// TIA Portal project "ModbusTCP_S7-1500" (V18)
// Test del protocolo Modbus TCP usando MB_Server y QModMaster

(* hardware
DEVICE "S7-1500/ET200MP station_1"  S7-1500 station
   slot 0: "Rail_0"  Rack  6ES7 590-1***0-0AA0
   slot 1: "PLC_1"  CPU 1511-1 PN  6ES7 511-1AL03-0AB0  V3.0
      slot 3: "CPU display_1"  6ES7591-1AA00-0AA0
      slot 32768: "PROFINET interface_1"  X1
         slot 32769: "Port_1"  X1 P1
         slot 32770: "Port_2"  X1 P2
      slot 34817: "Virtual CP interface port_1"  Virtual CP interface port  Virtual CP interface port
*)

// ===== PLC "PLC_1"  CPU 1511-1 PN =====

VAR_GLOBAL   // PLC tag table "Default tag table"
   "start" AT %I0.0 : Bool;
   "stop" AT %I0.1 : Bool;
   "motor" AT %Q0.0 : Bool;
   "System_Byte" AT %MB1 : Byte;
   "FirstScan" AT %M1.0 : Bool;
   "DiagStatusUpdate" AT %M1.1 : Bool;
   "AlwaysTRUE" AT %M1.2 : Bool;
   "AlwaysFALSE" AT %M1.3 : Bool;
   "System_Byte(1)" AT %MB1 : Byte;
   "Clock_Byte" AT %MB0 : Byte;
   "Clock_10Hz" AT %M0.0 : Bool;
   "Clock_5Hz" AT %M0.1 : Bool;
   "Clock_2.5Hz" AT %M0.2 : Bool;
   "Clock_2Hz" AT %M0.3 : Bool;
   "Clock_1.25Hz" AT %M0.4 : Bool;
   "Clock_1Hz" AT %M0.5 : Bool;
   "Clock_0.625Hz" AT %M0.6 : Bool;
   "Clock_0.5Hz" AT %M0.7 : Bool;
   "Alarma_1" AT %M100.0 : Bool;
   "Tag_1" AT %MW28 : Word;
   "Tag_2" AT %MW30 : Word;
   "Tag_3" AT %MW38 : Word;
   "Tag_4" AT %MW48 : Word;
   "Tag_5" AT %MW50 : Word;
   "Tag_6" AT %MW86 : Word;
   "Tag_7" AT %MW88 : Word;
   "Tag_8" AT %MW90 : Word;
END_VAR

DATA_BLOCK "Modbus_Data"   // DB1
{ S7_Optimized_Access := 'FALSE' }
VERSION : 0.1
   VAR
      Data_Array : Array[0..119] of UInt;
   END_VAR
BEGIN
   // Data_Array[52] : ALARMA W52: 0: Emergencia, 1: Térmico motor, 2: Falta fase
   // Data_Array[53] : ALARMA W53
   // Data_Array[54] : ALARMA W54
   // Data_Array[55] : ALARMA W55
END_DATA_BLOCK

DATA_BLOCK "Modbus_Config"   // DB2
{ S7_Optimized_Access := 'TRUE' }
VERSION : 0.1
   VAR
      Config : TCON_IP_v4;
   END_VAR
BEGIN
   Config.InterfaceId := 64;
   Config.ID := 16#1;
   Config.ConnectionType := 16#0B;
   Config.LocalPort := 502;
END_DATA_BLOCK

DATA_BLOCK "SCADA_Comm"   // DB4
{ S7_Optimized_Access := 'FALSE' }
VERSION : 0.1
   VAR
      cmd_Start : Bool;
      cmd_Stop : Bool;
      sts_Motor : Bool;
   END_VAR
BEGIN
END_DATA_BLOCK

DATA_BLOCK "FB_Alarmas1_DB"   // DB5
{ S7_Optimized_Access := 'TRUE' }
VERSION : 0.1
// stored: InstanceOfName FB_Alarmas
"FB_Alarmas"
BEGIN
END_DATA_BLOCK

DATA_BLOCK "FB_Alarmas2_DB"   // DB6
{ S7_Optimized_Access := 'TRUE' }
VERSION : 0.1
// stored: InstanceOfName FB_Alarmas
"FB_Alarmas"
BEGIN
END_DATA_BLOCK

DATA_BLOCK "FB_Sim_Produccion_DB"   // DB7
{ S7_Optimized_Access := 'TRUE' }
VERSION : 0.1
// stored: InstanceOfName FB_Sim_Produccion
"FB_Sim_Produccion"
BEGIN
END_DATA_BLOCK

DATA_BLOCK "FB_SIM_Produccion_V2_DB"   // DB8
{ S7_Optimized_Access := 'TRUE' }
VERSION : 0.1
// stored: InstanceOfName FB_SIM_Produccion_V2
"FB_SIM_Produccion_V2"
BEGIN
END_DATA_BLOCK

FUNCTION_BLOCK "FB_Alarmas"   // FB1, SCL
{ S7_Optimized_Access := 'TRUE' }
VERSION : 0.1
   VAR_INPUT
      i_Bit_0 : Bool;
      i_Bit_1 : Bool;
      i_Bit_2 : Bool;
      i_Bit_3 : Bool;
      i_Bit_4 : Bool;
      i_Bit_5 : Bool;
      i_Bit_6 : Bool;
      i_Bit_7 : Bool;
      i_Bit_8 : Bool;
      i_Bit_9 : Bool;
      i_Bit_10 : Bool;
      i_Bit_11 : Bool;
      i_Bit_12 : Bool;
      i_Bit_13 : Bool;
      i_Bit_14 : Bool;
      i_Bit_15 : Bool;
      i_Reset : Bool;   // Entrada del botón de reset
   END_VAR
   VAR_OUTPUT
      o_Bit_0 : Bool;
      o_Bit_1 : Bool;
      o_Bit_2 : Bool;
      o_Bit_3 : Bool;
      o_Bit_4 : Bool;
      o_Bit_5 : Bool;
      o_Bit_6 : Bool;
      o_Bit_7 : Bool;
      o_Bit_8 : Bool;
      o_Bit_9 : Bool;
      o_Bit_10 : Bool;
      o_Bit_11 : Bool;
      o_Bit_12 : Bool;
      o_Bit_13 : Bool;
      o_Bit_14 : Bool;
      o_Bit_15 : Bool;
      enAlarma : Bool;
   END_VAR
BEGIN
   // 1. Construcción de la palabra de alarmas actual
   // 3. Gestión de la salida
   // Si doy reset, la palabra de salida se pone a cero, sino refleja los bits de entrada.
   IF #i_Reset THEN
       // 1. Construcción de la palabra de alarmas actual
       #o_Bit_0 := 0;
       #o_Bit_1 := 0;
       #o_Bit_2 := 0;
       #o_Bit_3 := 0;
       #o_Bit_4 := 0;
       #o_Bit_5 := 0;
       #o_Bit_6 := 0;
       #o_Bit_7 := 0;
       #o_Bit_8 := 0;
       #o_Bit_9 := 0;
       #o_Bit_10 := 0;
       #o_Bit_11 := 0;
       #o_Bit_12 := 0;
       #o_Bit_13 := 0;
       #o_Bit_14 := 0;
       #o_Bit_15 := 0;
   ELSE
       // 1. Construcción de la palabra de alarmas actual
       #o_Bit_0 := #i_Bit_0;
       #o_Bit_1 := #i_Bit_1;
       #o_Bit_2 := #i_Bit_2;
       #o_Bit_3 := #i_Bit_3;
       #o_Bit_4 := #i_Bit_4;
       #o_Bit_5 := #i_Bit_5;
       #o_Bit_6 := #i_Bit_6;
       #o_Bit_7 := #i_Bit_7;
       #o_Bit_8 := #i_Bit_8;
       #o_Bit_9 := #i_Bit_9;
       #o_Bit_10 := #i_Bit_10;
       #o_Bit_11 := #i_Bit_11;
       #o_Bit_12 := #i_Bit_12;
       #o_Bit_13 := #i_Bit_13;
       #o_Bit_14 := #i_Bit_14;
       #o_Bit_15 := #i_Bit_15;
   END_IF;

   // Esto sigue siendo un poco largo pero es más limpio que un IF
   #enAlarma := #o_Bit_0 OR #o_Bit_1 OR #o_Bit_2 OR #o_Bit_3 OR
   #o_Bit_4 OR #o_Bit_5 OR #o_Bit_6 OR #o_Bit_7 OR
   #o_Bit_8 OR #o_Bit_9 OR #o_Bit_10 OR #o_Bit_11 OR
   #o_Bit_12 OR #o_Bit_13 OR #o_Bit_14 OR #o_Bit_15;

   // -------------------------------------------------------------
END_FUNCTION_BLOCK

FUNCTION_BLOCK "FB_Sim_Produccion"   // FB2, SCL
{ S7_Optimized_Access := 'TRUE' }
VERSION : 0.1
   VAR_INPUT
      IntervaloS : Time :=  T#1M;   // Intervalo de muestreo >> Escribe aquí T#1M o T#15M
   END_VAR
   VAR
      tCiclo : TON_TIME;   // Timer interno
      Seed : UDInt := 123456;   // Semilla aleatoria inicial
      Golpes : Int := 0;   // Estas variables son ESTÁTICAS: Se guardan solas en el DB de Instancia
   END_VAR
   VAR_TEMP
      valInt : Int;
   END_VAR
BEGIN
   // ============================================================
   // FB_Sim_Produccion — Versión Function Block (FB)
   // Simulación de datos de producción para SCADA Node3
   // ============================================================

   // 1. Temporizador cíclico
   #tCiclo(IN := NOT #tCiclo.Q, PT := #IntervaloS);

   // Lógica ejecutada en cada pulso del timer
   IF #tCiclo.Q THEN

       // --- SIMULACIÓN ALEATORIA ---

       // W14: TEMP_SP_SUP (180-220)
       #Seed := #Seed * 1664525 + 1013904223;
       #valInt := 180 + UDINT_TO_INT(#Seed MOD 41);
       "Tag_1" := #valInt;

       // W15: TEMP_SP_INF (160-200)
       #Seed := #Seed * 1664525 + 1013904223;
       #valInt := 160 + UDINT_TO_INT(#Seed MOD 41);
       "Tag_2" := #valInt;

       // W19: CONSUMO kW (10-25)
       #Seed := #Seed * 1664525 + 1013904223;
       #valInt := 10 + UDINT_TO_INT(#Seed MOD 16);
       "Tag_3" := #valInt;

       // W24: TEMP REAL SUP
       #Seed := #Seed * 1664525 + 1013904223;
       #valInt := 200 + UDINT_TO_INT(#Seed MOD 11) - 5;
       "Tag_4" := #valInt;

       // W25: TEMP REAL INF
       #Seed := #Seed * 1664525 + 1013904223;
       #valInt := 180 + UDINT_TO_INT(#Seed MOD 11) - 5;
       "Tag_5" := #valInt;

       // W43: ESTADO (0=Stop, 1=Run, 2=Alarma)
       #Seed := #Seed * 1664525 + 1013904223;
       #valInt := UDINT_TO_INT(#Seed MOD 3);
       "Tag_6" := #valInt;

       // W44: TIEMPO CICLO (8-12s)
       #Seed := #Seed * 1664525 + 1013904223;
       #valInt := 8 + UDINT_TO_INT(#Seed MOD 5);
       "Tag_7" := #valInt;

       // W45: CONTADOR GOLPES (Sumamos 5-20)
       #Seed := #Seed * 1664525 + 1013904223;
       #Golpes := #Golpes + 5 + UDINT_TO_INT(#Seed MOD 16);
       "Tag_8" := #Golpes;

   END_IF;
END_FUNCTION_BLOCK

FUNCTION_BLOCK "FB_SIM_Produccion_V2"   // FB3, SCL
{ S7_Optimized_Access := 'TRUE' }
VERSION : 0.1
   VAR_INPUT
      Enable : Bool := TRUE;
      IntervaloS : Time := T#1M;   // El contador suma cada este tiempo
   END_VAR
   VAR_OUTPUT
      outSPSup : Int;   // Conectar a W14 (%MW28)
      outSPInf : Int;   // Conectar a W15 (%MW30)
      outConsumo : Int;   // Conectar a W19 (%MW38)
      outTempSup : Int;   // Conectar a W24 (%MW48)
      outTempInf : Int;   // Conectar a W25 (%MW50)
      outCiclo : Int;   // Conectar a W44 (%MW88)
      outGolpes : Int;   // Conectar a W45 (%MW90)
   END_VAR
   VAR
      tCiclo : TON_TIME;   // Timer interno
      Seed : UDInt := 54321;   // Semilla aleatoria
      GolpesAcum : Int;   // Memoria interna de producción
      CicloUltimo : Int := 10;   // Valor inicial para que no empiece en 0
      PrimerScan : Bool := TRUE;
   END_VAR
   VAR_TEMP
      valInt : Int;
   END_VAR
BEGIN
   // ============================================================
   // FB_Sim_Produccion_V3 — Versión con Salidas Parametrizables
   // ============================================================
   (*
   Pin de Salida   Registro    Modbus PLC (Sugerido)  Descripción
   #outSPSup       W14 %MW28   SetPoint               Temp Superior
   outSPInf        W15 %MW30   SetPoint               Temp Inferior
   outConsumo      W19 %MW38   Consumo (kW)
   outTempSup      W24 %MW48   Temp Real Superior
   outTempInf      W25 %MW50   Temp Real Inferior
   outCiclo        W44 %MW88   Tiempo de Ciclo
   outGolpes       W45 %MW90   Contador de Producción
   *)

   // ============================================================
   // FB_Sim_Produccion_V7 — Versión Permanente (Salidas fijas)
   // ============================================================
   // 1. Temporizador
   #tCiclo(IN := #Enable AND NOT #tCiclo.Q,
           PT := #IntervaloS);

   IF NOT #Enable THEN
       RETURN;
   END_IF;

   // 2. CÁLCULO DE VALORES DINÁMICOS (Cada scan)
   #Seed := #Seed * 1664525 + 1013904223;

   #outSPSup := 200 + UDINT_TO_INT(#Seed MOD 3) - 1;
   #outSPInf := 180 + UDINT_TO_INT((#Seed / 10) MOD 3) - 1;
   #outTempSup := 198 + UDINT_TO_INT((#Seed / 100) MOD 5);
   #outTempInf := 178 + UDINT_TO_INT((#Seed / 1000) MOD 5);
   #outConsumo := 20 + UDINT_TO_INT((#Seed / 50) MOD 2);

   // 3. LÓGICA DE INCREMENTO (Solo cuando el timer da el pulso)
   IF #tCiclo.Q OR #PrimerScan THEN
       #GolpesAcum := #GolpesAcum + 1;
       #CicloUltimo := 8 + UDINT_TO_INT(#Seed MOD 5);
       #PrimerScan := FALSE;
   END_IF;

   // 4. ASIGNACIÓN PERMANENTE (Fuera del IF para que nunca sea cero)
   #outGolpes := #GolpesAcum;
   #outCiclo := #CicloUltimo;
END_FUNCTION_BLOCK

ORGANIZATION_BLOCK "Main"   // OB1, LAD, ProgramCycle
TITLE = "Main Program Sweep (Cycle)"
{ S7_Optimized_Access := 'TRUE' }
VERSION : 0.1
   VAR_INPUT
      Initial_Call : Bool;   // Initial call of this OB
      Remanence : Bool;   // =True, if remanent data are available
   END_VAR
   VAR_TEMP   // added for the SCL form of the ladder/FBD networks
      _w1 : Bool;
      _w2 : Bool;
   END_VAR
BEGIN

REGION Network 1: Configuracion basica MODBUS ( Nota con el IP: 0.0.0.0 ) asi escucha todo lo que llama
   // 1- Interfaz X1 del S7-1500 : 64   >>  16#40
   // 1- Conexion Type : TCP/IP  :  11 o 16#0B  , es igual
   // 3- Componente ID = 1
   // 4- Local Port  = 502
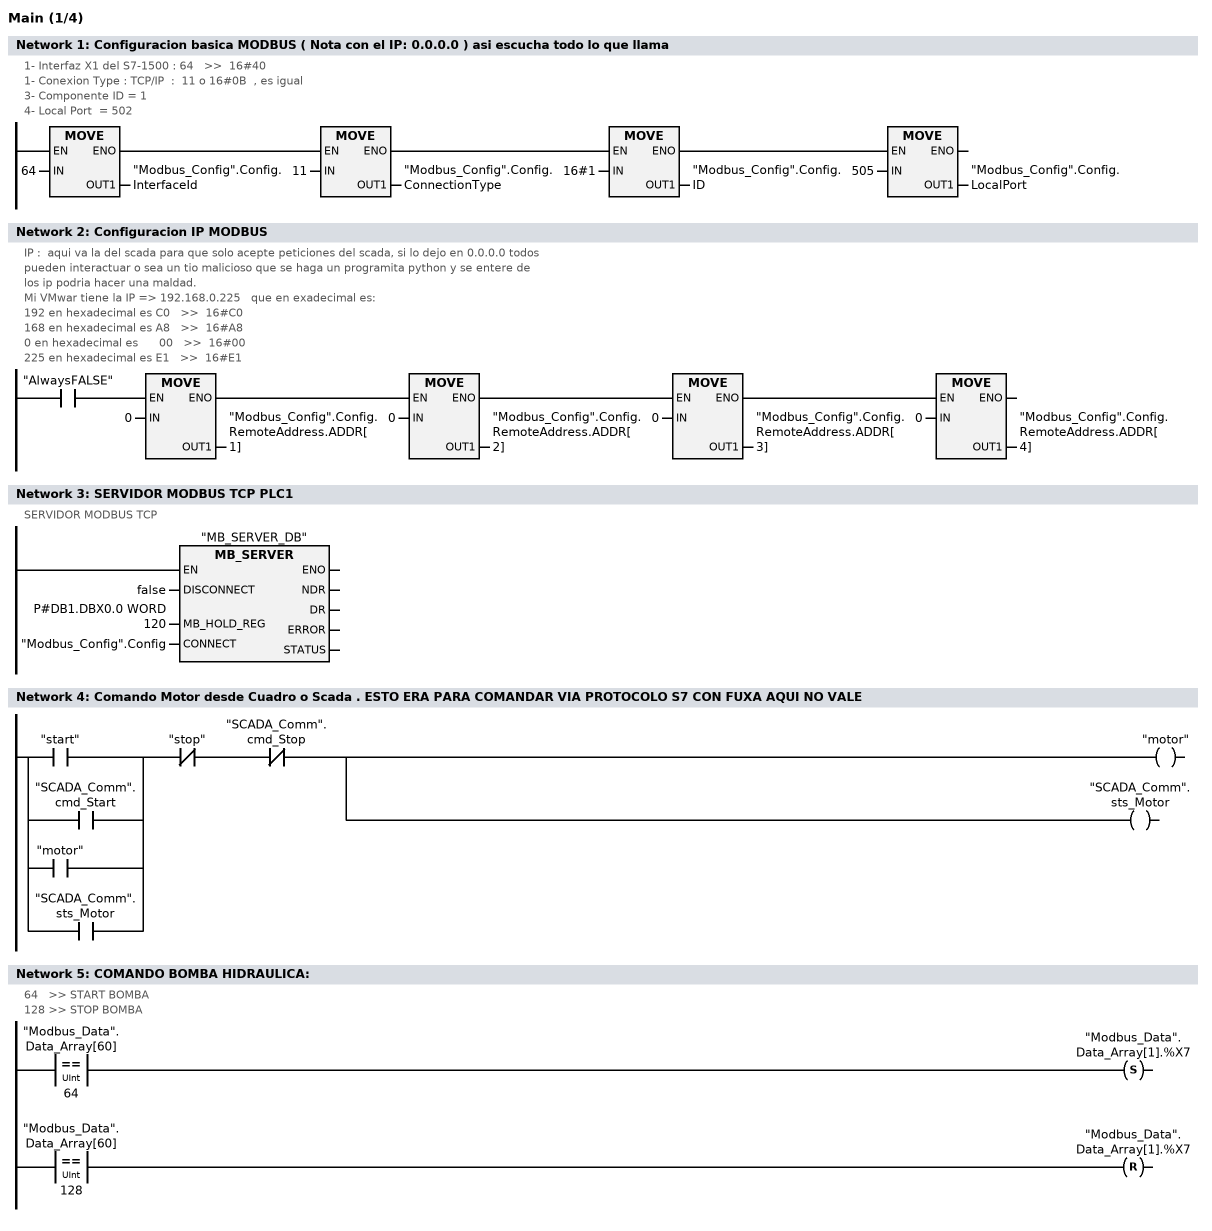
   RUNG wire#powerrail
      Move(in := 64, out1 => "Modbus_Config".Config.InterfaceId)
      Move(in := 11, out1 => "Modbus_Config".Config.ConnectionType)
      Move(in := 16#1, out1 => "Modbus_Config".Config.ID)
      Move(in := 505, out1 => "Modbus_Config".Config.LocalPort)
   END_RUNG
   // the same network as SCL:
   "Modbus_Config".Config.InterfaceId := 64;
   "Modbus_Config".Config.ConnectionType := 11;
   "Modbus_Config".Config.ID := 16#1;
   "Modbus_Config".Config.LocalPort := 505;
END_REGION

REGION Network 2: Configuracion IP MODBUS
   // IP :  aqui va la del scada para que solo acepte peticiones del scada, si lo dejo en 0.0.0.0 todos
   //       pueden interactuar o sea un tio malicioso que se haga un programita python y se entere de
   //       los ip podria hacer una maldad. 
   // 
   //      Mi VMwar tiene la IP => 192.168.0.225   que en exadecimal es:
   //         192 en hexadecimal es C0   >>  16#C0
   //         168 en hexadecimal es A8   >>  16#A8
   //         0 en hexadecimal es      00   >>  16#00
   //         225 en hexadecimal es E1   >>  16#E1
   RUNG wire#powerrail
      Contact( "AlwaysFALSE" )
      Move(in := 0, out1 => "Modbus_Config".Config.RemoteAddress.ADDR[1])
      Move(in := 0, out1 => "Modbus_Config".Config.RemoteAddress.ADDR[2])
      Move(in := 0, out1 => "Modbus_Config".Config.RemoteAddress.ADDR[3])
      Move(in := 0, out1 => "Modbus_Config".Config.RemoteAddress.ADDR[4])
   END_RUNG
   // the same network as SCL:
   IF "AlwaysFALSE" THEN
       "Modbus_Config".Config.RemoteAddress.ADDR[1] := 0;
       "Modbus_Config".Config.RemoteAddress.ADDR[2] := 0;
       "Modbus_Config".Config.RemoteAddress.ADDR[3] := 0;
       "Modbus_Config".Config.RemoteAddress.ADDR[4] := 0;
   END_IF;
END_REGION

REGION Network 3: SERVIDOR MODBUS TCP PLC1
   // SERVIDOR MODBUS TCP
   "MB_SERVER_DB"(DISCONNECT := false, MB_HOLD_REG := P#DB1.DBX0.0 WORD 120, CONNECT := "Modbus_Config".Config);   // MB_SERVER
END_REGION

REGION Network 4: Comando Motor desde Cuadro o Scada . ESTO ERA PARA COMANDAR VIA PROTOCOLO S7 CON FUXA AQUI NO VALE
   RUNG wire#powerrail
      Contact( "start" )
      wire#w1
      I_Contact( "stop" )
      I_Contact( "SCADA_Comm".cmd_Stop )
      wire#w2
      Coil( "motor" )
   END_RUNG
   RUNG wire#powerrail
      Contact( "SCADA_Comm".cmd_Start )
   END_RUNG wire#w1
   RUNG wire#powerrail
      Contact( "motor" )
   END_RUNG wire#w1
   RUNG wire#powerrail
      Contact( "SCADA_Comm".sts_Motor )
   END_RUNG wire#w1
   RUNG wire#w2
      Coil( "SCADA_Comm".sts_Motor )
   END_RUNG
   // the same network as SCL:
   "motor" := ("start" OR "SCADA_Comm".cmd_Start OR "motor" OR "SCADA_Comm".sts_Motor) AND NOT "stop" AND NOT "SCADA_Comm".cmd_Stop;
   "SCADA_Comm".sts_Motor := "motor";
END_REGION

REGION Network 5: COMANDO BOMBA HIDRAULICA:
   // 64   >> START BOMBA
   // 128 >> STOP BOMBA
   RUNG wire#powerrail
      { S7_Templates := "SrcType := UInt" } EQ_Contact(in1 := "Modbus_Data".Data_Array[60], in2 := 64)
      S_Coil( "Modbus_Data".Data_Array[1].%X7 )
   END_RUNG
   RUNG wire#powerrail
      { S7_Templates := "SrcType := UInt" } EQ_Contact(in1 := "Modbus_Data".Data_Array[60], in2 := 128)
      R_Coil( "Modbus_Data".Data_Array[1].%X7 )
   END_RUNG
   // the same network as SCL:
   IF "Modbus_Data".Data_Array[60] = 64 THEN "Modbus_Data".Data_Array[1].%X7 := TRUE; END_IF;
   IF "Modbus_Data".Data_Array[60] = 128 THEN "Modbus_Data".Data_Array[1].%X7 := FALSE; END_IF;
END_REGION

REGION Network 6: COMANDO RESISTENCIA:
   // 16   >> START
   // 32   >> STOP
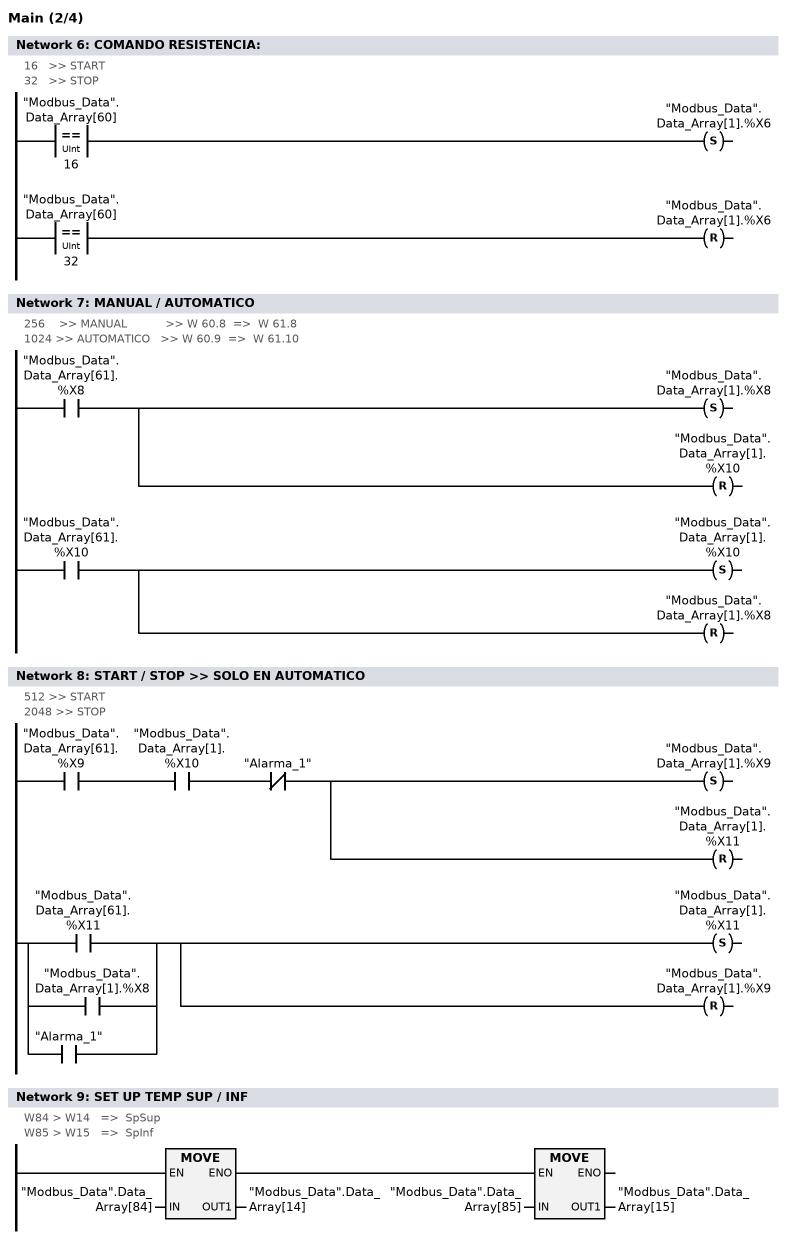
   RUNG wire#powerrail
      { S7_Templates := "SrcType := UInt" } EQ_Contact(in1 := "Modbus_Data".Data_Array[60], in2 := 16)
      S_Coil( "Modbus_Data".Data_Array[1].%X6 )
   END_RUNG
   RUNG wire#powerrail
      { S7_Templates := "SrcType := UInt" } EQ_Contact(in1 := "Modbus_Data".Data_Array[60], in2 := 32)
      R_Coil( "Modbus_Data".Data_Array[1].%X6 )
   END_RUNG
   // the same network as SCL:
   IF "Modbus_Data".Data_Array[60] = 16 THEN "Modbus_Data".Data_Array[1].%X6 := TRUE; END_IF;
   IF "Modbus_Data".Data_Array[60] = 32 THEN "Modbus_Data".Data_Array[1].%X6 := FALSE; END_IF;
END_REGION

REGION Network 7: MANUAL / AUTOMATICO
   // 256    >> MANUAL           >> W 60.8  =>  W 61.8
   // 1024 >> AUTOMATICO   >> W 60.9  =>  W 61.10
   RUNG wire#powerrail
      Contact( "Modbus_Data".Data_Array[61].%X8 )
      wire#w1
      S_Coil( "Modbus_Data".Data_Array[1].%X8 )
   END_RUNG
   RUNG wire#w1
      R_Coil( "Modbus_Data".Data_Array[1].%X10 )
   END_RUNG
   RUNG wire#powerrail
      Contact( "Modbus_Data".Data_Array[61].%X10 )
      wire#w2
      S_Coil( "Modbus_Data".Data_Array[1].%X10 )
   END_RUNG
   RUNG wire#w2
      R_Coil( "Modbus_Data".Data_Array[1].%X8 )
   END_RUNG
   // the same network as SCL:
   #_w1 := "Modbus_Data".Data_Array[61].%X8;
   IF #_w1 THEN
       "Modbus_Data".Data_Array[1].%X8 := TRUE;
       "Modbus_Data".Data_Array[1].%X10 := FALSE;
   END_IF;
   #_w2 := "Modbus_Data".Data_Array[61].%X10;
   IF #_w2 THEN
       "Modbus_Data".Data_Array[1].%X10 := TRUE;
       "Modbus_Data".Data_Array[1].%X8 := FALSE;
   END_IF;
END_REGION

REGION Network 8: START / STOP >> SOLO EN AUTOMATICO
   // 512 >> START
   // 2048 >> STOP
   RUNG wire#powerrail
      Contact( "Modbus_Data".Data_Array[61].%X9 )
      Contact( "Modbus_Data".Data_Array[1].%X10 )
      I_Contact( "Alarma_1" )
      wire#w1
      S_Coil( "Modbus_Data".Data_Array[1].%X9 )
   END_RUNG
   RUNG wire#w1
      R_Coil( "Modbus_Data".Data_Array[1].%X11 )
   END_RUNG
   RUNG wire#powerrail
      Contact( "Modbus_Data".Data_Array[61].%X11 )
      wire#w2
      S_Coil( "Modbus_Data".Data_Array[1].%X11 )
   END_RUNG
   RUNG wire#powerrail
      Contact( "Modbus_Data".Data_Array[1].%X8 )
   END_RUNG wire#w2
   RUNG wire#powerrail
      Contact( "Alarma_1" )
   END_RUNG wire#w2
   RUNG wire#w2
      R_Coil( "Modbus_Data".Data_Array[1].%X9 )
   END_RUNG
   // the same network as SCL:
   #_w1 := "Modbus_Data".Data_Array[61].%X9 AND "Modbus_Data".Data_Array[1].%X10 AND NOT "Alarma_1";
   IF #_w1 THEN
       "Modbus_Data".Data_Array[1].%X9 := TRUE;
       "Modbus_Data".Data_Array[1].%X11 := FALSE;
   END_IF;
   #_w2 := "Modbus_Data".Data_Array[61].%X11 OR "Modbus_Data".Data_Array[1].%X8 OR "Alarma_1";
   IF #_w2 THEN
       "Modbus_Data".Data_Array[1].%X11 := TRUE;
       "Modbus_Data".Data_Array[1].%X9 := FALSE;
   END_IF;
END_REGION

REGION Network 9: SET UP TEMP SUP / INF
   // W84 > W14   =>  SpSup
   // W85 > W15   =>  SpInf
   RUNG wire#powerrail
      Move(in := "Modbus_Data".Data_Array[84], out1 => "Modbus_Data".Data_Array[14])
      Move(in := "Modbus_Data".Data_Array[85], out1 => "Modbus_Data".Data_Array[15])
   END_RUNG
   // the same network as SCL:
   "Modbus_Data".Data_Array[14] := "Modbus_Data".Data_Array[84];
   "Modbus_Data".Data_Array[15] := "Modbus_Data".Data_Array[85];
END_REGION

REGION Network 10 (SCL): RECETAS: W62 a W76 >> W2 a W15 + W27 -----> Ver la Tabla Estado en el ScadaNode
   // Ricete  Spessore
   // RECETA_EMPUJE
   // RECETA_DISPARO
   // RECETA_EXPANSION
   // RECETA_2DO_EMPUJE
   // RECETA_2DO_DISPARO
   // RECETA_2DO_EXPANSION
   // Duracion Limpieza Dosificacion
   // Retraso Limpieza Dosificacion
   // Retraso subida plato central doble ciclo
   // Vaso
   // Ciclos de limpieza de la dosificacion
   // Temperatura de consigna superior
   // Temperatura de consigna inferior
   // Numero de formas en el molde
   // Mover recetas: W62 a W76  >>  W2 a W15 + W27
   "Modbus_Data".Data_Array[2] := "Modbus_Data".Data_Array[62];
   "Modbus_Data".Data_Array[3] := "Modbus_Data".Data_Array[63];
   "Modbus_Data".Data_Array[4] := "Modbus_Data".Data_Array[64];
   "Modbus_Data".Data_Array[5] := "Modbus_Data".Data_Array[65];
   "Modbus_Data".Data_Array[6] := "Modbus_Data".Data_Array[66];
   "Modbus_Data".Data_Array[7] := "Modbus_Data".Data_Array[67];
   "Modbus_Data".Data_Array[8] := "Modbus_Data".Data_Array[68];
   "Modbus_Data".Data_Array[9] := "Modbus_Data".Data_Array[69];
   "Modbus_Data".Data_Array[10] := "Modbus_Data".Data_Array[70];
   "Modbus_Data".Data_Array[11] := "Modbus_Data".Data_Array[71];
   "Modbus_Data".Data_Array[12] := "Modbus_Data".Data_Array[72];
   "Modbus_Data".Data_Array[13] := "Modbus_Data".Data_Array[73];
   "Modbus_Data".Data_Array[14] := "Modbus_Data".Data_Array[74];
   "Modbus_Data".Data_Array[15] := "Modbus_Data".Data_Array[75];

   // Registro final al destino especial
   "Modbus_Data".Data_Array[27] := "Modbus_Data".Data_Array[76];
END_REGION

REGION Network 11: ALARMAS >> W52
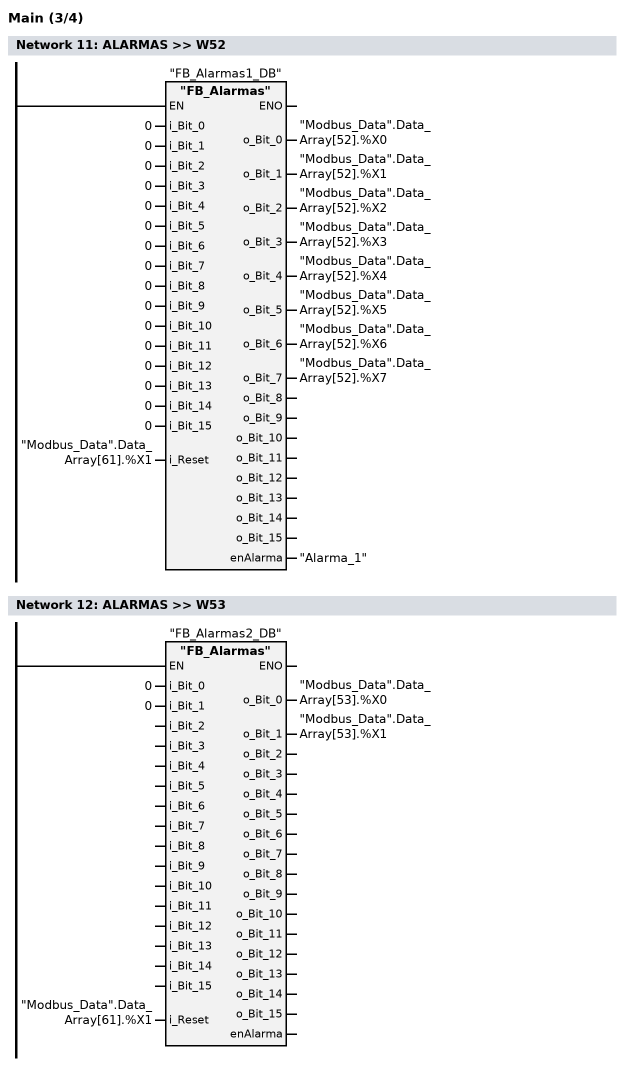
   RUNG wire#powerrail
      "FB_Alarmas1_DB"(i_Bit_0 := 0, i_Bit_1 := 0, i_Bit_2 := 0, i_Bit_3 := 0, i_Bit_4 := 0, i_Bit_5 := 0, i_Bit_6 := 0, i_Bit_7 := 0, i_Bit_8 := 0, i_Bit_9 := 0, i_Bit_10 := 0, i_Bit_11 := 0, i_Bit_12 := 0, i_Bit_13 := 0, i_Bit_14 := 0, i_Bit_15 := 0, i_Reset := "Modbus_Data".Data_Array[61].%X1, o_Bit_0 => "Modbus_Data".Data_Array[52].%X0, o_Bit_1 => "Modbus_Data".Data_Array[52].%X1, o_Bit_2 => "Modbus_Data".Data_Array[52].%X2, o_Bit_3 => "Modbus_Data".Data_Array[52].%X3, o_Bit_4 => "Modbus_Data".Data_Array[52].%X4, o_Bit_5 => "Modbus_Data".Data_Array[52].%X5, o_Bit_6 => "Modbus_Data".Data_Array[52].%X6, o_Bit_7 => "Modbus_Data".Data_Array[52].%X7, o_Bit_8 =>, o_Bit_9 =>, o_Bit_10 =>, o_Bit_11 =>, o_Bit_12 =>, o_Bit_13 =>, o_Bit_14 =>, o_Bit_15 =>, enAlarma => "Alarma_1")
   END_RUNG
   // the same network as SCL:
   "FB_Alarmas1_DB"(i_Bit_0 := 0,   // "FB_Alarmas"
                    i_Bit_1 := 0,
                    i_Bit_2 := 0,
                    i_Bit_3 := 0,
                    i_Bit_4 := 0,
                    i_Bit_5 := 0,
                    i_Bit_6 := 0,
                    i_Bit_7 := 0,
                    i_Bit_8 := 0,
                    i_Bit_9 := 0,
                    i_Bit_10 := 0,
                    i_Bit_11 := 0,
                    i_Bit_12 := 0,
                    i_Bit_13 := 0,
                    i_Bit_14 := 0,
                    i_Bit_15 := 0,
                    i_Reset := "Modbus_Data".Data_Array[61].%X1,
                    o_Bit_0 => "Modbus_Data".Data_Array[52].%X0,
                    o_Bit_1 => "Modbus_Data".Data_Array[52].%X1,
                    o_Bit_2 => "Modbus_Data".Data_Array[52].%X2,
                    o_Bit_3 => "Modbus_Data".Data_Array[52].%X3,
                    o_Bit_4 => "Modbus_Data".Data_Array[52].%X4,
                    o_Bit_5 => "Modbus_Data".Data_Array[52].%X5,
                    o_Bit_6 => "Modbus_Data".Data_Array[52].%X6,
                    o_Bit_7 => "Modbus_Data".Data_Array[52].%X7,
                    enAlarma => "Alarma_1");
END_REGION

REGION Network 12: ALARMAS >> W53
   RUNG wire#powerrail
      "FB_Alarmas2_DB"(i_Bit_0 := 0, i_Bit_1 := 0, i_Bit_2 :=, i_Bit_3 :=, i_Bit_4 :=, i_Bit_5 :=, i_Bit_6 :=, i_Bit_7 :=, i_Bit_8 :=, i_Bit_9 :=, i_Bit_10 :=, i_Bit_11 :=, i_Bit_12 :=, i_Bit_13 :=, i_Bit_14 :=, i_Bit_15 :=, i_Reset := "Modbus_Data".Data_Array[61].%X1, o_Bit_0 => "Modbus_Data".Data_Array[53].%X0, o_Bit_1 => "Modbus_Data".Data_Array[53].%X1, o_Bit_2 =>, o_Bit_3 =>, o_Bit_4 =>, o_Bit_5 =>, o_Bit_6 =>, o_Bit_7 =>, o_Bit_8 =>, o_Bit_9 =>, o_Bit_10 =>, o_Bit_11 =>, o_Bit_12 =>, o_Bit_13 =>, o_Bit_14 =>, o_Bit_15 =>, enAlarma =>)
   END_RUNG
   // the same network as SCL:
   "FB_Alarmas2_DB"(i_Bit_0 := 0,   // "FB_Alarmas"
                    i_Bit_1 := 0,
                    i_Reset := "Modbus_Data".Data_Array[61].%X1,
                    o_Bit_0 => "Modbus_Data".Data_Array[53].%X0,
                    o_Bit_1 => "Modbus_Data".Data_Array[53].%X1);
END_REGION

REGION Network 13: SIMULA PRODUCCION
   // Pin de Salida   Registro    Modbus PLC (Sugerido)  Descripción
   // ==========   ======    ==================  ==========
   // outSPSup          W14 %MW28    SetPoint               Temp Superior
   // outSPInf             W15 %MW30   SetPoint                Temp Inferior
   // outConsumo    W19 %MW38   Consumo (kW)
   // outTempSup    W24 %MW48   Temp Real Superior
   // outTempInf       W25 %MW50   Temp Real Inferior
   // outCiclo             W44 %MW88   Tiempo de Ciclo
   // outGolpes         W45 %MW90   Contador de Producción
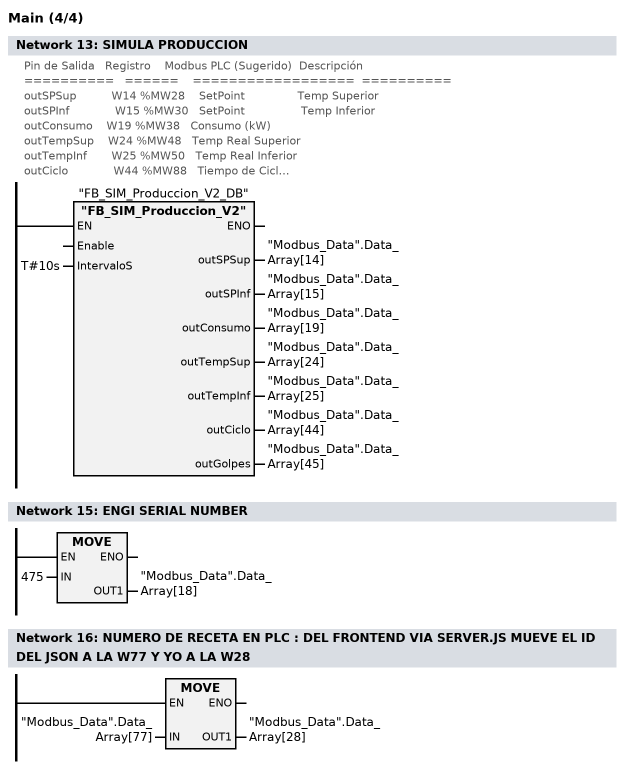
   RUNG wire#powerrail
      "FB_SIM_Produccion_V2_DB"(Enable :=, IntervaloS := T#10s, outSPSup => "Modbus_Data".Data_Array[14], outSPInf => "Modbus_Data".Data_Array[15], outConsumo => "Modbus_Data".Data_Array[19], outTempSup => "Modbus_Data".Data_Array[24], outTempInf => "Modbus_Data".Data_Array[25], outCiclo => "Modbus_Data".Data_Array[44], outGolpes => "Modbus_Data".Data_Array[45])
   END_RUNG
   // the same network as SCL:
   "FB_SIM_Produccion_V2_DB"(IntervaloS := T#10s,   // "FB_SIM_Produccion_V2"
                           outSPSup => "Modbus_Data".Data_Array[14],
                           outSPInf => "Modbus_Data".Data_Array[15],
                           outConsumo => "Modbus_Data".Data_Array[19],
                           outTempSup => "Modbus_Data".Data_Array[24],
                           outTempInf => "Modbus_Data".Data_Array[25],
                           outCiclo => "Modbus_Data".Data_Array[44],
                           outGolpes => "Modbus_Data".Data_Array[45]);
END_REGION

REGION Network 14 (SCL): ESTADO DE LA MAQUINA
   // 0- DESCONOCIDO, 1- MANUAL , 2- AUTOMATICO, 3- ALARMA
   // // Lógica de Estados para SCADA (STATO_MACCHINA - W43)

    IF "Alarma_1" THEN
   //     //"STATO_MACCHINA" := 3; // ESTADO 3: ALARMA (Rojo)
        "Modbus_Data".Data_Array[43] := 3;
    ELSIF "Modbus_Data".Data_Array[1].%X10 THEN
   //     //"STATO_MACCHINA" := 2; // ESTADO 2: AUTOMÁTICO (Verde)
        "Modbus_Data".Data_Array[43] := 2;
    ELSIF "Modbus_Data".Data_Array[1].%X8 THEN
   //     //"STATO_MACCHINA" := 1; // ESTADO 1: MANUAL (Azul)
        "Modbus_Data".Data_Array[43] := 1;
    ELSE
   //     //"STATO_MACCHINA" := 0; // ESTADO 1: DESCONOCIDO
        "Modbus_Data".Data_Array[43] := 0;
   END_IF;
END_REGION

REGION Network 15: ENGI SERIAL NUMBER
   RUNG wire#powerrail
      Move(in := 475, out1 => "Modbus_Data".Data_Array[18])
   END_RUNG
   // the same network as SCL:
   "Modbus_Data".Data_Array[18] := 475;
END_REGION

REGION Network 16: NUMERO DE RECETA EN PLC : DEL FRONTEND VIA SERVER.JS MUEVE EL ID DEL JSON A LA W77 Y YO A LA W28
   RUNG wire#powerrail
      Move(in := "Modbus_Data".Data_Array[77], out1 => "Modbus_Data".Data_Array[28])
   END_RUNG
   // the same network as SCL:
   "Modbus_Data".Data_Array[28] := "Modbus_Data".Data_Array[77];
END_REGION
END_ORGANIZATION_BLOCK